FUNCTION_BLOCK FB_SensorNODecoratorTest EXTENDS FB_SensorDecoratorTestParent 
VAR
	
END_VAR

(*			
	EVERDE sp. z o.o.
	Rafał Osajda		05.02.2025		TC 4026.13		wer. 0.0.0.1
	Zwraca aktualny stan czujnika
*)
METHOD IsActive : BOOL
IsActive			:= THIS^.bContactTest;
END_METHOD

END_FUNCTION_BLOCK

(* stored: Version 1.1.0.1
   POU FB_SensorNODecoratorTest: Id {2db5dc4b-91ae-401b-8c31-39e5d116893b}, SpecialFunc None
   Method IsActive: Id {bee729fc-1548-4ad7-8b73-4f8b865f8d90} *)
